Universal Robots PolyScope program: robotics-project.urp

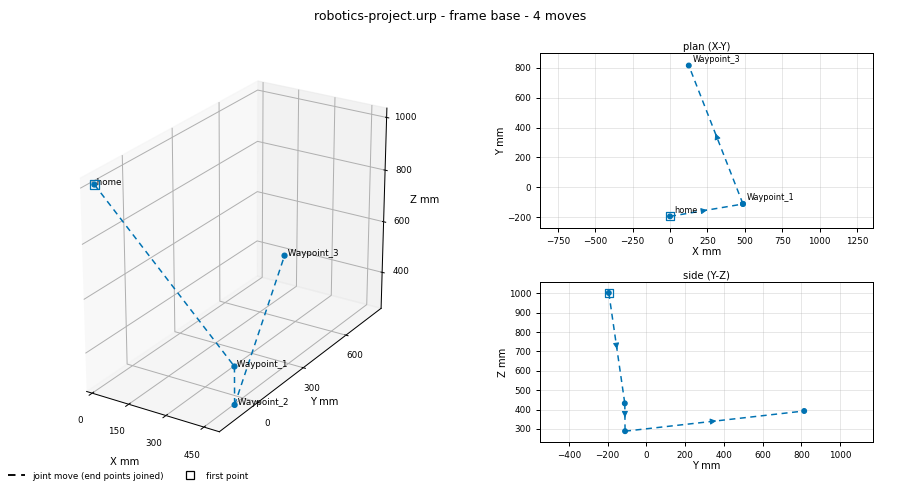
[picture p0: tool path of robotics-project.urp in frame base, 4 of 4 moves have a stored position in this frame; points joined in program order, loops and branches not executed]
Program robotics-project (createdIn=3.4.4.412 lastSavedIn=3.4.4.412 directory=/programs installation=default robotSerialNumber=2017356443)
Calibrated DH parameters: a=[0.000092, -0.116521, -0.182101, -0.000106, 0.000044, 0]; d=[0.089391, 255.189113, -82.629387, -172.449369, 0.094782, 0.082637]; alpha=[1.569598, 0.001603, 0.002015, 1.570234, -1.570307, 0]; deltaTheta=[-0.000017, 1.293309, -0.204843, -1.088417, 0.000036, -0.000078]
Robot Program (runOnlyOnce=false motionType=MoveJ speed=1.047198 acceleration=1.396263 useActiveTCP=false)
  Script: rq_close_and_wait(1)
  Script: rq_open_and_wait(1)
  MoveJ speed 60 deg/s, acceleration 80 deg/s^2 (useActiveTCP=false)
    Waypoint home: TCP in base x=-0.084 y=-193.553 z=1001.627 mm, rx=-0.0012 ry=-2.2231 rz=2.2182 rad; joints [0, -90, 0, -90, 0, 0] deg; flange x=-0.152 y=-193.553 z=1001.627 mm, rx=-0.0015 ry=-2.2232 rz=2.2183 rad
  MoveJ speed 60 deg/s, acceleration 80 deg/s^2 (useActiveTCP=false)
    Waypoint Waypoint_1: TCP in base x=487.141 y=-111.118 z=432.1 mm, rx=2.2183 ry=-2.2241 rz=0.0014 rad; joints [-0.004, -89.996, -90.003, -90.007, 89.989, -0.01] deg
    Waypoint Waypoint_2: TCP in base x=486.767 y=-109.777 z=288.556 mm, rx=-2.1588 ry=2.1572 rz=-0.1356 rad; joints [0.152, -92.934, -110.379, -59.604, 89.986, -0.015] deg
  URCap Gripper (Robotiq_2-Finger_Adaptive_Gripper, Robotiq Inc.) data=position = 100
    | force = 0
    | speed = 0
    | blocking = true
    | slaveIds = [9]
  MoveJ speed 60 deg/s, acceleration 80 deg/s^2 (useActiveTCP=false)
    Waypoint Waypoint_3: TCP in base x=125.169 y=814.03 z=392.743 mm, rx=0.0094 ry=1.1715 rz=2.894 rad; joints [89.049, -134.523, -44.521, -135, -90, 0] deg
  URCap Gripper (Robotiq_2-Finger_Adaptive_Gripper, Robotiq Inc.) data=position = 0
    | force = 0
    | speed = 0
    | blocking = true
    | slaveIds = [9]
